// TwinCAT 3 PLC project fee_rix_motion
// ProgramVersion: 3.1.4022.7
// libraries:
//   LCLS General, * (SLAC)
//   lcls-twincat-motion, * (SLAC)
//   lcls2-cc-lib, * (SLAC)
//   Tc2_Standard, * (Beckhoff Automation GmbH)
//   Tc2_System, * (Beckhoff Automation GmbH)
//   Tc3_Module, * (Beckhoff Automation GmbH)
// project tree:
//   GVLs/ Main.TcGVL (not stored)
//   / PlcTask.TcTTO (not stored)
//   POUs/ PRG_1_PlcTask.TcPOU, PRG_2_PMPS_PRE.TcPOU (not stored), PRG_3_PMPS_POST.TcPOU (not stored), PRG_IM1K1_PPM.TcPOU, PRG_IM2K1_PPM.TcPOU (not stored), PRG_ST1K1_ZOS.TcPOU (not stored)
// real-time tasks:
//   TASK PlcTask: cycle T#10ms, priority 20, ADS port 350
// motion (NC):
//   TASK NC-Task 1 SAF: cycle T#1ms, priority 4, ADS port 501
//   TASK NC-Task 1 SVB: cycle T#10ms, priority 8, ADS port 511
//   AXIS Axis 1 IM1K1-PPM-MMS (id 1)
//     Dynamic: AccelerationMaximum=200, DecelerationMaximum=200, Acceleration=200, Deceleration=200, Jerk=500, DelayTime=0.004
//     Velo: Maximum=65
//     TargetPosControl: Range=0.002, Time=2
//     OtherSettings: AllowMotionCmdToSlave=true
//     encoder EncType=29
//       EncPara: ScaleFactorNumerator=5e-05, Offset=-214686.941, MaxCount=#xffffffff, ReferenceSystem=1
//         SoftEndMinControl: Enable=true, Range=-100
//         SoftEndMaxControl: Enable=true, Range=-8.82
//     drive DrvType=24
//       Analog: VeloReferenz=100, ScaleFactorActTorque=0.1
//       TimeComp: TaskDelayCycles=1
//     controller CtrType=2
//       CtrPara: PriorControlFactor=1
//         PosDiffControl: Range=1
//         PID: PosKp=20, PosExtKp=1, PosExtVelo=0.1, DeadBandPosition=0.002
//         Observer: BandWidth=20
//   AXIS Axis 2 IM2K1-PPM-MMS (id 2)
//     Dynamic: AccelerationMaximum=200, DecelerationMaximum=200, Acceleration=200, Deceleration=200, Jerk=500, DelayTime=0.004
//     Velo: Maximum=65
//     TargetPosControl: Range=0.002, Time=2
//     OtherSettings: AllowMotionCmdToSlave=true
//     encoder EncType=29
//       EncPara: ScaleFactorNumerator=5e-05, Offset=-214686.941, MaxCount=#xffffffff, ReferenceSystem=1
//         SoftEndMinControl: Range=-100
//         SoftEndMaxControl: Range=-9.09
//     drive DrvType=24
//       Analog: VeloReferenz=100, ScaleFactorActTorque=0.1
//       TimeComp: TaskDelayCycles=1
//     controller CtrType=2
//       CtrPara: PriorControlFactor=1
//         PosDiffControl: Range=1
//         PID: PosKp=20, PosExtKp=1, PosExtVelo=0.1, DeadBandPosition=0.002
//         Observer: BandWidth=20
//   AXIS Axis 3 ST1K1-ZOS-MMS (id 3)
//     OtherSettings: AllowMotionCmdToSlave=true
//     encoder EncType=1
//     drive DrvType=5
//       Analog: ScaleFactorActTorque=0.1
//     controller CtrType=1
//       CtrPara: PriorControlFactor=1
//         Observer: BandWidth=20
// I/O:
//   DEVICE PLC Rail (EtherCAT), AmsNetId 134.79.82.163.2.1
//     Power (EK1200)
//     EtherCAT Panel (EK1100)
// variable links:
//   fee_rix_motion Instance <-> PLC Rail (EtherCAT)/EtherCAT Panel (EK1100)/EC E1 (EK1122)/X1 IM1K1-PPM (EK1100)/IM1K1-EL2004
//     PlcTask Outputs/Main.M1.bBrakeRelease <-> Channel 1/Output
//     PlcTask Outputs/PRG_IM1K1_PPM.fbIM1K1.fbGige.bGigePower <-> Channel 2/Output
//   fee_rix_motion Instance <-> PLC Rail (EtherCAT)/EtherCAT Panel (EK1100)/EC E1 (EK1122)/X1 IM1K1-PPM (EK1100)/IM1K1-EL3062
//     PlcTask Inputs/PRG_IM1K1_PPM.fbIM1K1.fbPowerMeter.iVoltageINT <-> AI Standard Channel 1/Value
//   fee_rix_motion Instance <-> PLC Rail (EtherCAT)/EtherCAT Panel (EK1100)/EC E1 (EK1122)/X1 IM1K1-PPM (EK1100)/IM1K1-EL3314
//     PlcTask Inputs/PRG_IM1K1_PPM.fbIM1K1.fbPowerMeter.fbThermoCouple.bError <-> TC Inputs Channel 1/Status/Error
//     PlcTask Inputs/PRG_IM1K1_PPM.fbIM1K1.fbPowerMeter.fbThermoCouple.bOverrange <-> TC Inputs Channel 1/Status/Overrange
//     PlcTask Inputs/PRG_IM1K1_PPM.fbIM1K1.fbPowerMeter.fbThermoCouple.bUnderrange <-> TC Inputs Channel 1/Status/Underrange
//     PlcTask Inputs/PRG_IM1K1_PPM.fbIM1K1.fbPowerMeter.fbThermoCouple.iRaw <-> TC Inputs Channel 1/Value
//     PlcTask Inputs/PRG_IM1K1_PPM.fbIM1K1.fbYagThermoCouple.bError <-> TC Inputs Channel 2/Status/Error
//     PlcTask Inputs/PRG_IM1K1_PPM.fbIM1K1.fbYagThermoCouple.bOverrange <-> TC Inputs Channel 2/Status/Overrange
//     PlcTask Inputs/PRG_IM1K1_PPM.fbIM1K1.fbYagThermoCouple.bUnderrange <-> TC Inputs Channel 2/Status/Underrange
//     PlcTask Inputs/PRG_IM1K1_PPM.fbIM1K1.fbYagThermoCouple.iRaw <-> TC Inputs Channel 2/Value
//   fee_rix_motion Instance <-> PLC Rail (EtherCAT)/EtherCAT Panel (EK1100)/EC E1 (EK1122)/X1 IM1K1-PPM (EK1100)/IM1K1-EL4004
//     PlcTask Outputs/PRG_IM1K1_PPM.fbIM1K1.fbGige.iIlluminatorINT <-> AO Outputs Channel 1/Analog output
//   fee_rix_motion Instance <-> PLC Rail (EtherCAT)/EtherCAT Panel (EK1100)/EC E1 (EK1122)/X1 IM1K1-PPM (EK1100)/IM1K1-EL7041
//     PlcTask Inputs/Main.M1.bLimitBackwardEnable <-> STM Status/Status/Digital input 2
//     PlcTask Inputs/Main.M1.bLimitForwardEnable <-> STM Status/Status/Digital input 1
//   fee_rix_motion Instance <-> PLC Rail (EtherCAT)/EtherCAT Panel (EK1100)/EC E1 (EK1122)/X2 IM2K1-PPM (EK1100)/IM2K1-EL2004
//     PlcTask Outputs/Main.M2.bBrakeRelease <-> Channel 1/Output
//     PlcTask Outputs/PRG_IM2K1_PPM.fbIM2K1.fbGige.bGigePower <-> Channel 2/Output
//   fee_rix_motion Instance <-> PLC Rail (EtherCAT)/EtherCAT Panel (EK1100)/EC E1 (EK1122)/X2 IM2K1-PPM (EK1100)/IM2K1-EL3062
//     PlcTask Inputs/PRG_IM2K1_PPM.fbIM2K1.fbPowerMeter.iVoltageINT <-> AI Standard Channel 1/Value
//   fee_rix_motion Instance <-> PLC Rail (EtherCAT)/EtherCAT Panel (EK1100)/EC E1 (EK1122)/X2 IM2K1-PPM (EK1100)/IM2K1-EL3314
//     PlcTask Inputs/PRG_IM2K1_PPM.fbIM2K1.fbPowerMeter.fbThermoCouple.bError <-> TC Inputs Channel 1/Status/Error
//     PlcTask Inputs/PRG_IM2K1_PPM.fbIM2K1.fbPowerMeter.fbThermoCouple.bOverrange <-> TC Inputs Channel 1/Status/Overrange
//     PlcTask Inputs/PRG_IM2K1_PPM.fbIM2K1.fbPowerMeter.fbThermoCouple.bUnderrange <-> TC Inputs Channel 1/Status/Underrange
//     PlcTask Inputs/PRG_IM2K1_PPM.fbIM2K1.fbPowerMeter.fbThermoCouple.iRaw <-> TC Inputs Channel 1/Value
//     PlcTask Inputs/PRG_IM2K1_PPM.fbIM2K1.fbYagThermoCouple.bError <-> TC Inputs Channel 2/Status/Error
//     PlcTask Inputs/PRG_IM2K1_PPM.fbIM2K1.fbYagThermoCouple.bOverrange <-> TC Inputs Channel 2/Status/Overrange
//     PlcTask Inputs/PRG_IM2K1_PPM.fbIM2K1.fbYagThermoCouple.bUnderrange <-> TC Inputs Channel 2/Status/Underrange
//     PlcTask Inputs/PRG_IM2K1_PPM.fbIM2K1.fbYagThermoCouple.iRaw <-> TC Inputs Channel 2/Value
//   fee_rix_motion Instance <-> PLC Rail (EtherCAT)/EtherCAT Panel (EK1100)/EC E1 (EK1122)/X2 IM2K1-PPM (EK1100)/IM2K1-EL4004
//     PlcTask Outputs/PRG_IM2K1_PPM.fbIM2K1.fbGige.iIlluminatorINT <-> AO Outputs Channel 1/Analog output
//   fee_rix_motion Instance <-> PLC Rail (EtherCAT)/EtherCAT Panel (EK1100)/EC E1 (EK1122)/X2 IM2K1-PPM (EK1100)/IM2K1-EL7041
//     PlcTask Inputs/Main.M2.bLimitBackwardEnable <-> STM Status/Status/Digital input 2
//     PlcTask Inputs/Main.M2.bLimitForwardEnable <-> STM Status/Status/Digital input 1
//   fee_rix_motion Instance <-> NC-Task 1 SAF/Axes/Axis 1 IM1K1-PPM-MMS
//     PlcTask Inputs/Main.M1.Axis.NcToPlc <-> Outputs/ToPlc
//     PlcTask Outputs/Main.M1.Axis.PlcToNc <-> Inputs/FromPlc
//   fee_rix_motion Instance <-> NC-Task 1 SAF/Axes/Axis 2 IM2K1-PPM-MMS
//     PlcTask Inputs/Main.M2.Axis.NcToPlc <-> Outputs/ToPlc
//     PlcTask Outputs/Main.M2.Axis.PlcToNc <-> Inputs/FromPlc

// ---- POUs/PRG_1_PlcTask.TcPOU
PROGRAM PRG_1_PlcTask
VAR
END_VAR

PRG_2_PMPS_PRE();

// STUFF HERE

PRG_3_PMPS_POST();

END_PROGRAM

// ---- POUs/PRG_IM1K1_PPM.TcPOU
PROGRAM PRG_IM1K1_PPM
VAR
    {attribute 'pytmc' := '
        pv: IM1K1:PPM
        io: io
    '}
    {attribute 'TcLinkTo' := '.fbGige.iIlluminatorINT := TIIB[IM1K1-EL4004]^AO Outputs Channel 1^Analog output;
                              .fbGige.bGigePower := TIIB[IM1K1-EL2004]^Channel 2^Output;
                              .fbPowerMeter.iVoltageINT := TIIB[IM1K1-EL3062]^AI Standard Channel 1^Value;
                              .fbPowerMeter.fbThermoCouple.bError := TIIB[IM1K1-EL3314]^TC Inputs Channel 1^Status^Error;
                              .fbPowerMeter.fbThermoCouple.bUnderrange := TIIB[IM1K1-EL3314]^TC Inputs Channel 1^Status^Underrange;
                              .fbPowerMeter.fbThermoCouple.bOverrange := TIIB[IM1K1-EL3314]^TC Inputs Channel 1^Status^Overrange;
                              .fbPowerMeter.fbThermoCouple.iRaw := TIIB[IM1K1-EL3314]^TC Inputs Channel 1^Value;
                              .fbYagThermoCouple.bError := TIIB[IM1K1-EL3314]^TC Inputs Channel 2^Status^Error;
                              .fbYagThermoCouple.bUnderrange := TIIB[IM1K1-EL3314]^TC Inputs Channel 2^Status^Underrange;
                              .fbYagThermoCouple.bOverrange := TIIB[IM1K1-EL3314]^TC Inputs Channel 2^Status^Overrange;
                              .fbYagThermoCouple.iRaw := TIIB[IM1K1-EL3314]^TC Inputs Channel 2^Value'}
    fbIM1K1: FB_PPM;
END_VAR

fbIM1K1(
    stYStage := Main.M1,
    fPolished := -71.92,
    fFrosted := -97.93, // Actually a second polished yag
    fPower := -47.92,
    fOut := -8.82);

END_PROGRAM
